Fanuc KAREL source: kb00107.KL

-- PROVISIONAL review KL for V1013-1; original PC SHA256 8d390345de0f385d535bac66fcdac5652cc4f1418e4e9cb3e115eba28184111a
-- Incomplete behavior may be omitted. Consult companion uncertainty JSON. Do not deploy.
PROGRAM KB00107
%NOLOCKGROUP
VAR
  RESULT : BOOLEAN
-- UNRESOLVED_DECL P1 type=000106
BEGIN
  -- UNRESOLVED_PC offsets 5-28; opcodes 27,22,1C,27,9D,76,23
  -- UNRESOLVED_PC offsets 33-37; opcodes 7F
END KB00107
